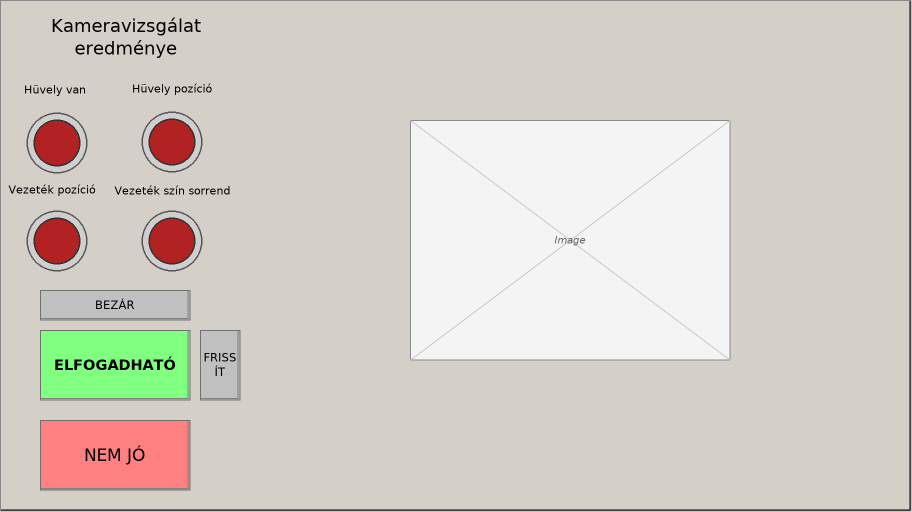
VISUALIZATION Kamera  // 912x512
    Rectangle (0,0 910x510)
    Button (40,420 150x70), "NEM JÓ", invisible if: GVL.bNTCEredmenyGombokRejtve
        OnMouseUp: execute {
            GVL.bNTCKameraNemJo:=TRUE;
            GVL.bNTCEredmenyGombokRejtve:=TRUE;
            GVL.bKameraEredmenyekRejtve:=TRUE;
        }
    Label (10,80 90x20), "Hüvely van"
    Lamp1 (22,108 70x70), variable: GVL.bKameraHulseVanOK, style: Lamp-Lamp1-Green
    Lamp1 (22,108 70x70), variable: NOT GVL.bKameraHulseVanOK, invisible if: NOT KAMERA.bVizsgalatKesz OR GVL.bKameraHulseVanOK, style: Lamp-Lamp1-Red
    Lamp1 (137,107 70x70), variable: GVL.bKameraHulsePozOK, style: Lamp-Lamp1-Green
    Lamp1 (137,206 70x70), variable: GVL.bKameraSzinekOK, style: Lamp-Lamp1-Green
    Label (108,181 129x20), "Vezeték szín sorrend"
    Label (130,80 84x18), "Hüvely pozíció"
    Lamp1 (137,107 70x70), variable: NOT GVL.bKameraHulsePozOK, invisible if: NOT KAMERA.bVizsgalatKesz OR GVL.bKameraHulsePozOK, style: Lamp-Lamp1-Red
    Lamp1 (137,206 70x70), variable: NOT GVL.bKameraSzinekOK, invisible if: NOT KAMERA.bVizsgalatKesz OR GVL.bKameraSzinekOK, style: Lamp-Lamp1-Red
    Label (0,180 104x20), "Vezeték pozíció"
    Lamp1 (22,206 70x70), variable: GVL.bKameraVezetekPozOK, style: Lamp-Lamp1-Green
    Lamp1 (22,206 70x70), variable: NOT GVL.bKameraVezetekPozOK, invisible if: NOT KAMERA.bVizsgalatKesz OR GVL.bKameraVezetekPozOK, style: Lamp-Lamp1-Red
    Label (51,10 150x54), "Kameravizsgálat eredménye"
    Button (40,330 150x70), "ELFOGADHATÓ", invisible if: GVL.bNTCEredmenyGombokRejtve
        OnMouseUp: execute {
            GVL.bNTCKameraElfogadva:=TRUE;
            GVL.bNTCEredmenyGombokRejtve:=TRUE;
            GVL.bKameraEredmenyekRejtve:=TRUE;
        }
    Button (40,290 150x30), "BEZÁR", invisible if: GVL.bNTCBezarGombRejtve
        OnMouseUp: execute {
            //GVL.bNTCBezarGombRejtve:=TRUE;
            GVL.bKameraEredmenyekRejtve:=TRUE;
        }
    Button (200,330 40x70), "FRISSÍT"
        OnMouseUp: execute { GVL.iBitmap_Version:= GVL.iBitmap_Version+1; }
    Image (410,120 320x240)
        p871682116: GVL.iBitmap_Version
        p84334746: GVL.sNTCKameraImageID
END_VISUALIZATION

(* stored: Version 1.1.0.1, ProductVersion 3.1.4024.11
   Visu Kamera: Id {a7eab427-6190-4c1e-9278-f5ba0c6c90b0} *)
